FUNCTION_BLOCK EL3161
VAR
	_io : EL3xx1_Data;
	{attribute addProperty Name "WcState"}
	_wcState : WcStateInputToggle;
	{attribute addProperty Name "Info data"}
	_infoData : InfoDataAds;
END_VAR

PROPERTY IO : REFERENCE TO EL3xx1_Data
GET
IO REF= _io;
END_GET
END_PROPERTY

PROPERTY WcState : REFERENCE TO WcStateInputToggle
GET
WcState REF= _wcState;
END_GET
END_PROPERTY

END_FUNCTION_BLOCK

(* stored: Version 1.1.0.1, ProductVersion 3.1.4024.9
   POU EL3161: Id {b44205dc-e3da-0afc-3b4e-b4e5f00259e8}, SpecialFunc None
   Property IO: Id {56100f2d-7d85-055e-20b5-d0c3565597f7}
   Get Get: Id {1dfe978c-825b-0864-174f-3a83c81ace3f}
   Property WcState: Id {8ea55574-7f51-0d81-282c-97a467b43a21}
   Get Get: Id {2eb4f738-9bc7-0d69-0f88-377203063eb4} *)
